Staubli VAL3: setByteAt.pgx

public program setByteAt(num x_nByteIndex, num x_nByte, num& x_nBuffer[])
  local num l_nHIword
  local num l_nLOword
  local string l_sBinWord
  local string l_sTempBinByte
begin

  //Header begin

  //This function is trivial, it just set to "x_nByte" the "x_nByteIndex" element of the array x_nBuffer.
  //
  //Input parameters
  //
  //num x_nByteIndex: the index of the element in the "x_nBuffer[]" array representing the byte we want to read.
	//num x_nRes: the byte value we want to set.
  //
  //Output parameters
  //
  //num x_nBuffer[1]: the monodimensional array of num where we are writing a byte (most likely a plc's memory area we are about to write with writeArea).
  //
  //Examples
  //
  //call S7:setWordAt(0,231,l_nLocalByte)
  //
  //History
  // Creation: 24-12-16 - Alessio Villa
  //Header end

  if x_nByte<0 or x_nByte>255
    x_nBuffer[x_nByteIndex]=0
  endIf

  x_nBuffer[x_nByteIndex]=x_nByte

end
